FUNCTION_BLOCK CentralController (* Basic Function Block Type *)
  (* Standard: 61499-2 *)
  (* Version 0.0, 1/14/2024, midxav, Template *)
  PACKAGE Main;
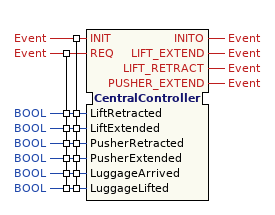
  EVENT_INPUT
    INIT WITH LiftRetracted, LiftExtended, PusherRetracted, PusherExtended, LuggageArrived, LuggageLifted; (* Initialization Request *)
    REQ WITH LiftRetracted, LiftExtended, PusherRetracted, PusherExtended, LuggageArrived, LuggageLifted; (* Normal Execution Request *)
  END_EVENT
  EVENT_OUTPUT
    INITO; (* Initialization Confirm *)
    LIFT_EXTEND;
    LIFT_RETRACT;
    PUSHER_EXTEND;
  END_EVENT
  VAR_INPUT
    LiftRetracted : BOOL; (* Input event qualifier *)
    LiftExtended : BOOL;
    PusherRetracted : BOOL;
    PusherExtended : BOOL;
    LuggageArrived : BOOL;
    LuggageLifted : BOOL;
  END_VAR
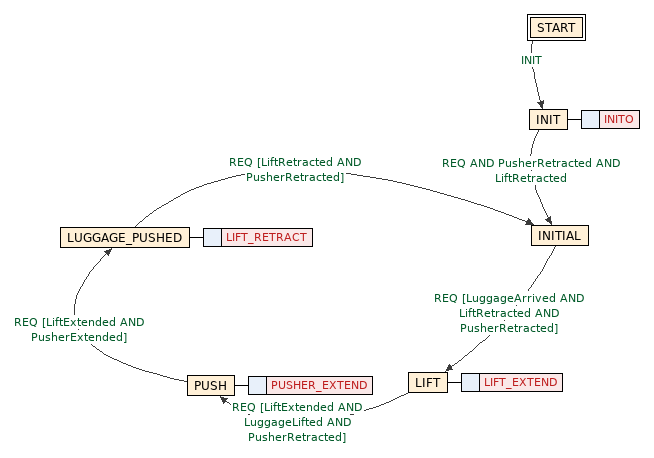
  EC_STATES
    START; (* Initial State *)
    INIT : -> INITO; (* Initialization *)
    INITIAL;
    LIFT : -> LIFT_EXTEND;
    PUSH : -> PUSHER_EXTEND;
    LUGGAGE_PUSHED : -> LIFT_RETRACT;
  END_STATES
  EC_TRANSITIONS
    START TO INIT := INIT;
    INIT TO INITIAL := REQ AND PusherRetracted AND LiftRetracted;
    INITIAL TO LIFT := REQ [LuggageArrived AND LiftRetracted AND PusherRetracted];
    LIFT TO PUSH := REQ [LiftExtended AND LuggageLifted AND PusherRetracted];
    PUSH TO LUGGAGE_PUSHED := REQ [LiftExtended AND PusherExtended];
    LUGGAGE_PUSHED TO INITIAL := REQ [LiftRetracted AND PusherRetracted];
  END_TRANSITIONS
END_FUNCTION_BLOCK
